Staubli VAL3: test.pgx

program test(screen& x_scr)
  local num l_nItem
  local string sold[4]
begin
  call changeValue(x_scr,l_nItem,0,4,5,5,sTab)
end
